PROGRAM Read_Payload
VAR
	EL3061_Lead_Bit AT %I* 	: INT;
	EL3061_Rear_Bit AT %I* 	: INT;
	
	//axle of lead trailer
	R3_Bit			: REAL;
	R3_BitTare		: REAL := 8043;
	R31_BitPerTon	: REAL := 7.8864; //bit caused by payload on lead trailer
	R32_BitPerTon	: REAL := 7.8864; //bit caused by payload on rear trailer
	
	//axle of rear trailer
	R4_Bit			: REAL;
	R4_BitTare		: REAL := 8043;
	R42_BitPerTon	: REAL := 7.8864;
	
	Payload_Lead	: REAL;
	Payload_Rear	: REAL;
	Payload_Total	: REAL;	
	
	Threshold_Lead	: REAL := 40.5;
	Threshold_Rear	: REAL := 72;	
	Overload_Lead	: BOOL := FALSE;
	Overload_Rear	: BOOL := FALSE;
END_VAR

R3_Bit := INT_TO_REAL(EL3061_Lead_Bit);
R4_Bit := INT_TO_REAL(EL3061_Rear_Bit);

(*
Payload_Rear	:= (R4_Bit - R4_BitTare) / R42_BitPerTon;
Payload_Lead	:= (R3_Bit - (R32_BitPerTon * Payload_Rear)) / R31_BitPerTon;
Payload_Total	:= Payload_Lead + Payload_Rear;
*)

//Payload_Rear	:= (R4_Bit - R4_BitTare) / R42_BitPerTon;

IF GVL.Lead_Trailer_State = 8 OR GVL.Lead_Trailer_State = 17416 THEN
	Payload_Lead	:= R3_Bit;
ELSE
	Payload_Lead	:= 0;
END_IF

IF GVL.Rear_Trailer_State = 8 THEN
	Payload_Rear	:= R4_Bit;
ELSE
	Payload_Rear	:= 0;
END_IF
Payload_Rear	:= R4_Bit;

IF Payload_Lead < 0 THEN
	Payload_Lead := 0;
END_IF

IF Payload_Rear < 0 THEN
	Payload_Rear := 0;
END_IF

IF Payload_Lead > Threshold_Lead THEN
	Overload_Lead := TRUE;
ELSE
	Overload_Lead := FALSE;	
END_IF

IF Payload_Rear > Threshold_Rear THEN
	Overload_Rear := TRUE;
ELSE
	Overload_Rear := FALSE;	
END_IF

(*
IF Read_GPS.Speed < 1 AND Background_IMU.Pitch < 3 AND Background_IMU.Roll < 3 THEN
	Payload	:= Payload_Raw;
END_IF

(* check for overload *)
IF Payload > Threshold THEN
	Overload := TRUE;
ELSE
	Overload := FALSE;	
END_IF
*)

END_PROGRAM

(* stored: Version 1.1.0.1, ProductVersion 3.1.4024.6
   POU Read_Payload: Id {54a58c0d-9bb6-4287-ad4a-87a5313c1987}, SpecialFunc None *)
